Staubli VAL3: readMe.pgx

public program readMe()
begin
  //
  //
  //
end
